/// Window Tracking action
INTERFACE I_TrackingActionListener EXTENDS __System.IQueryInterface

METHOD M_ActionZoneChangedEvent
VAR_INPUT
	mZoneIndex	: UINT; // Deleted zone index
	mZoneData	: ST_WindowTrackingZone; // Data of deleted zone
END_VAR
END_METHOD

/// Zone deleted
METHOD M_ActionZoneDeletedEvent
VAR_INPUT
	mZoneIndex	: UINT; // Deleted zone index
	mZoneData	: ST_WindowTrackingZone; // Data of deleted zone
END_VAR
END_METHOD

END_INTERFACE

(* stored: Version 1.1.0.1, ProductVersion 3.1.4020.6
   Itf I_TrackingActionListener: Id {31080e27-a665-4d70-b9e5-39da84d7c529}
   Method M_ActionZoneChangedEvent: Id {d74eaf57-8370-4154-aced-4b78d6a5e4fe}
   Method M_ActionZoneDeletedEvent: Id 218015ec-b14b-41e1-a1b6-70282250ba4d *)
